FUNCTION_BLOCK FB_SimulatedDigIn IMPLEMENTS ITF_DigIn
VAR
	internalState : BOOL;
END_VAR

METHOD get : BOOL
VAR_INPUT
END_VAR
get := internalState;
END_METHOD

END_FUNCTION_BLOCK

(* stored: Version 1.1.0.1, ProductVersion 3.1.4026.8
   POU FB_SimulatedDigIn: Id {387a2786-04b8-428a-9692-51d1a64f4124}, SpecialFunc None
   Method get: Id {ab4738cb-7b7e-4807-b9e1-d626a405b4f7} *)
